(* PLC project 117_1_V0.5.project, CODESYS CODESYS V3.5 SP17 Patch 3 *)
(* stored: creationDateTime 1970-01-01T00:00:00, modificationDateTime 2026-03-26T18:14:32.4070562 *)

FUNCTION_BLOCK InputManager
  VAR
    InputBytes : ARRAY[0..1] OF BYTE;  (* Физические входы *)
    bitsInput : ARRAY[0..15] OF BOOL;  (* Логический массив битов *)
    iByte : INT;
    iBit : INT;
    inputReals : ARRAY[tenza1000kgSensor..(lastAnalogInIndex - 1)] OF REAL;
  END_VAR

            FOR iByte := 0 TO 1 DO
    FOR iBit := 0 TO 7 DO
        bitsInput[iByte*8 + iBit] := (InputBytes[iByte] AND SHL(BYTE#16#01, iBit)) <> 0;
    END_FOR
END_FOR
          

METHOD get_discrete_data : BOOL
  VAR_INPUT
    varName : ALL_DI;
  END_VAR
                  get_discrete_data := bitsInput[varName];
                
END_METHOD
END_FUNCTION_BLOCK
